{attribute 'GeneratedUsingTerminal: KL1302'}
{attribute addProperty BoxType "KL1302"}
{attribute addProperty Description ""}
{attribute addProperty Physics ""}
{attribute addProperty Id "Channel_1AT %I*Channel_87C95E760Channel_2AT %I*Channel_87C95E760"}
{attribute addProperty CRC "3141065359"}
{attribute addProperty Size "0"}
TYPE KL1302_BB38DA8F :
STRUCT
	{attribute addProperty Name "Channel_1"}
	Channel_1 : Channel_87C95E76;
	{attribute addProperty Name "Channel_2"}
	Channel_2 : Channel_87C95E76;
END_STRUCT
END_TYPE

(* stored: Version 1.2.0.0, ProductVersion 3.1.4024.11
   DUT KL1302_BB38DA8F: Id {b2aebbe3-0eb1-4336-a351-109b14c8f88b} *)
